// TIA Portal V15.1 export
// export: Created 2024-05-17T05:38:10.6995703Z, ExportSetting WithDefaults, DisplayName Totally Integrated Automation Portal, DisplayVersion V15.1 Update 5, DisplayName TIA Portal Openness, DisplayVersion V15.1 Update 5, DisplayName SINAMICS Startdrive Advanced, DisplayVersion V15.1, DisplayName G130, G150, S120, S150, SINAMICS MV, S210, DisplayVersion V15.1, DisplayName G110M, G120, G120C, G120D, G120P, DisplayVersion V15.1, DisplayName STEP 7 Professional, DisplayVersion V15.1 Update 5, DisplayName STEP 7 Safety, DisplayVersion V15.1, DisplayName WinCC Professional, DisplayVersion V15.1 Update 5, DisplayName SIMATIC Visualization Architect, DisplayVersion V15.1
DATA_BLOCK "_209000AE01JC31"   // DB1117
{ S7_Optimized_Access := 'TRUE' }
AUTHOR : VCC
FAMILY : AlarmHnd
VERSION : 0.1
// stored: AutoNumber false, DBAccessibleFromOPCUA true, InstanceOfName LETAFuseCPC20PN, InstanceOfType FB
"LETAFuseCPC20PN"
   // VAR_INPUT
   //    I_NewShift { ExternalAccessible := 'False'; ExternalVisible := 'False'; ExternalWritable := 'False'} : Bool;
   //    I_EnableAlarm { ExternalAccessible := 'False'; ExternalVisible := 'False'; ExternalWritable := 'False'} : Bool;
   //    C_HWInput { ExternalAccessible := 'False'; ExternalVisible := 'False'; ExternalWritable := 'False'} : HW_IO;
   //    C_Block1_TotalCurrent { ExternalAccessible := 'False'; ExternalVisible := 'False'; ExternalWritable := 'False'} : HW_IO;
   //    C_Block1_StatusControl { ExternalAccessible := 'False'; ExternalVisible := 'False'; ExternalWritable := 'False'} : HW_IO;
   //    "C_Block1_MeasurementU/I" { ExternalAccessible := 'False'; ExternalVisible := 'False'; ExternalWritable := 'False'} : HW_IO;
   //    C_Block2_TotalCurrent { ExternalAccessible := 'False'; ExternalVisible := 'False'; ExternalWritable := 'False'} : HW_IO;
   //    C_Block2_StatusControl { ExternalAccessible := 'False'; ExternalVisible := 'False'; ExternalWritable := 'False'} : HW_IO;
   //    "C_Block2_MeasurementU/I" { ExternalAccessible := 'False'; ExternalVisible := 'False'; ExternalWritable := 'False'} : HW_IO;
   //    C_Config { ExternalAccessible := 'False'; ExternalVisible := 'False'; ExternalWritable := 'False'} : "ETAFuseCPC20PNConfig";
   // END_VAR
   // VAR_OUTPUT
   //    O_AlarmABCondition { ExternalAccessible := 'False'; ExternalVisible := 'False'; ExternalWritable := 'False'} : Bool;
   //    O_AlarmA { ExternalAccessible := 'False'; ExternalVisible := 'False'; ExternalWritable := 'False'} : Bool;
   //    O_AlarmB { ExternalAccessible := 'False'; ExternalVisible := 'False'; ExternalWritable := 'False'} : Bool;
   //    O_AlarmC { ExternalAccessible := 'False'; ExternalVisible := 'False'; ExternalWritable := 'False'} : Bool;
   //    O_AlarmD { ExternalAccessible := 'False'; ExternalVisible := 'False'; ExternalWritable := 'False'} : Bool;
   //    H_AlarmDWord { ExternalAccessible := 'False'; ExternalVisible := 'False'; ExternalWritable := 'False'} : DWord;
   // END_VAR
   // VAR_IN_OUT
   //    IO_ETAFuseData : "ETAFuseData";
   //    H_HMI : "H_HMI";
   //    H_ETAFuseCPC20PN : "H_ETAFuseCPC20PN";
   // END_VAR
   // VAR
   //    AC_StatusCPC20_Bit0 { ExternalAccessible := 'False'; ExternalVisible := 'False'; ExternalWritable := 'False'} : Bool;
   //    AC_StatusCPC20_Bit1 { ExternalAccessible := 'False'; ExternalVisible := 'False'; ExternalWritable := 'False'} : Bool;
   //    AC_StatusCPC20_Bit4 { ExternalAccessible := 'False'; ExternalVisible := 'False'; ExternalWritable := 'False'} : Bool;
   //    AC_StatusCPC20_Bit7 { ExternalAccessible := 'False'; ExternalVisible := 'False'; ExternalWritable := 'False'} : Bool;
   //    AC_StatusCPC20_Bit9 { ExternalAccessible := 'False'; ExternalVisible := 'False'; ExternalWritable := 'False'} : Bool;
   //    AC_StatusCPC20_Bit10 { ExternalAccessible := 'False'; ExternalVisible := 'False'; ExternalWritable := 'False'} : Bool;
   //    AC_ReadNomCurr { ExternalAccessible := 'False'; ExternalVisible := 'False'; ExternalWritable := 'False'} : Bool;
   //    AlarmABCondition { ExternalAccessible := 'False'; ExternalVisible := 'False'; ExternalWritable := 'False'} : Bool;
   //    AlarmA { ExternalAccessible := 'False'; ExternalVisible := 'False'; ExternalWritable := 'False'} : Bool;
   //    AlarmB { ExternalAccessible := 'False'; ExternalVisible := 'False'; ExternalWritable := 'False'} : Bool;
   //    AlarmC { ExternalAccessible := 'False'; ExternalVisible := 'False'; ExternalWritable := 'False'} : Bool;
   //    AlarmD { ExternalAccessible := 'False'; ExternalVisible := 'False'; ExternalWritable := 'False'} : Bool;
   //    ReadNominalCurrentActive { ExternalAccessible := 'False'; ExternalVisible := 'False'; ExternalWritable := 'False'} : Bool;
   //    EnableAlarm { ExternalAccessible := 'False'; ExternalVisible := 'False'; ExternalWritable := 'False'} : Bool;
   // END_VAR
   // VAR RETAIN
   //    H_ReadNomCurr { ExternalAccessible := 'False'; ExternalVisible := 'False'; ExternalWritable := 'False'} : Bool;
   //    H_CancelReadNomCurr { ExternalAccessible := 'False'; ExternalVisible := 'False'; ExternalWritable := 'False'} : Bool;
   // END_VAR
   // VAR
   //    H_UpChannel { ExternalAccessible := 'False'; ExternalVisible := 'False'; ExternalWritable := 'False'} : Bool;
   //    H_DownChannel { ExternalAccessible := 'False'; ExternalVisible := 'False'; ExternalWritable := 'False'} : Bool;
   //    H_SwitchON { ExternalAccessible := 'False'; ExternalVisible := 'False'; ExternalWritable := 'False'} : Bool;
   //    H_SwitchOFF { ExternalAccessible := 'False'; ExternalVisible := 'False'; ExternalWritable := 'False'} : Bool;
   //    H_Transfer { ExternalAccessible := 'False'; ExternalVisible := 'False'; ExternalWritable := 'False'} : Bool;
   //    H_Reset { ExternalAccessible := 'False'; ExternalVisible := 'False'; ExternalWritable := 'False'} : Bool;
   //    _ETAFuseCPC20PNSub { ExternalAccessible := 'False'; ExternalVisible := 'False'; ExternalWritable := 'False'} : "LETAFuseCPC20PNSub";
   //    T_ResetControl { ExternalAccessible := 'False'; ExternalVisible := 'False'; ExternalWritable := 'False'} : TON_TIME;
   //    T_EnableAlarm { ExternalAccessible := 'False'; ExternalVisible := 'False'; ExternalWritable := 'False'} : TON_TIME;
   //    Edge { ExternalAccessible := 'False'; ExternalVisible := 'False'; ExternalWritable := 'False'} : Array[0..10] of Bool;
   // END_VAR
BEGIN
END_DATA_BLOCK
